// TwinCAT 3 PLC project PLC
// ProgramVersion: 3.1.4024.0
// libraries:
//   Tc2_Standard, * (Beckhoff Automation GmbH)
//   Tc2_System, * (Beckhoff Automation GmbH)
//   Tc3_Module, * (Beckhoff Automation GmbH)
// project tree:
//   / PlcTask.TcTTO
//   POUs/ MAIN.TcPOU, TankControl01.TcPOU, TankControl02.TcPOU
//   POUs/Simulation/ IntegralCalculate.TcPOU, Scale.TcPOU, Simulation.TcPOU, TankLevelSimulator.TcPOU
// real-time tasks:
//   TASK PlcTask: cycle T#10ms, priority 20, ADS port 350

CONFIGURATION PLC
    RESOURCE PLC ON TwinCAT3
        TASK PlcTask(INTERVAL := T#10ms, PRIORITY := 20);
        PROGRAM MAIN WITH PlcTask : MAIN;
    END_RESOURCE
END_CONFIGURATION

// ---- POUs/MAIN.TcPOU
PROGRAM MAIN
VAR
	TankControl01				: TankControl01;
	Enable						: BOOL;
	TempReq						: REAL := 22.0;
	VolReq						: REAL := 1.2;
	TankDiam					: REAL := 1.0;
	TankHeight					: REAL := 10;
	LevelSensor					: WORD;
	TempSensor					: WORD;
	StartControl				: BOOL;
	FillValve					: BOOL;
	EmptyValve					: BOOL;
	HeatValve					: BOOL;
	
	Temp						: REAL;
	MixerMotor: BOOL;
END_VAR

Simulation(TankDiam := TankDiam, FillValve := TankControl01.FillValveCmd, HeatValve := TankControl01.HeatValveCmd, EmptyValve := TankControl01.EmptyValveCmd);
TankControl01(
    Enable := Enable,
    TemperatureReq := TempReq,
    VolumeReq := VolReq,
    TankDiameter := TankDiam,
    TankHeight := TankHeight,
    LevelSensor := TO_WORD(Simulation.Level),
    TemperatureSensor := TO_WORD(Simulation.Temperature),
    StartControl := StartControl);
FillValve := TankControl01.FillValveCmd;
EmptyValve := TankControl01.EmptyValveCmd;
HeatValve := TankControl01.HeatValveCmd;
MixerMotor := TankControl01.MixerMotorCmd;
// LevelSensor: input not connected
// TempSensor: input not connected

END_PROGRAM

// ---- POUs/TankControl01.TcPOU
FUNCTION_BLOCK TankControl01
VAR_INPUT
	Enable				:	BOOL;		// enable
	TemperatureReq		:	REAL;		// temperature request
	VolumeReq			:	REAL;		// volume request
	TankDiameter		:	REAL;		
	TankHeight			:	REAL;
	LevelSensor			:	WORD;		// raw value from AI
	TemperatureSensor	:	WORD;		// raw value from AI
	StartControl		:	BOOL;		// start tank control
END_VAR
VAR_OUTPUT
	FillValveCmd		:	BOOL;		// valve to fill the tank
	EmptyValveCmd		:	BOOL;		// valve to empty the tank
	HeatValveCmd		:	BOOL;		// valve to heat the tank
	MixerMotorCmd		:	BOOL;		// mixer motor inside tank
END_VAR
VAR
	LevelScaled			: 	REAL;
	TemperatureScaled	: 	REAL;
	TankVolume			: 	REAL;
	CalculationsOK		:	BOOL;
	SeqStep				:	(START, FILL, HEAT, EMPTY) := START;
END_VAR

(*
When Start Control switch is activated , Fill Valve opens and liquid fills the tank.
When liquid reaches the requested level, Fill Valve closes. 
Then Heat Valve opens and heats up the liquid. 
When the liquid inside the tank reaches the requested temperature, Empty Valve opens to empty the tank.
Mixer Motor ensures stirring during the heating process.
*)

IF Enable THEN
	SetSequence();
	SetOutput();
END_IF

METHOD Calculations : BOOL
VAR_INPUT

END_VAR

VAR
	HeightTotal			: REAL;
	LevelDoneOk			: BOOL;
	VolumeDoneOk		: BOOL;
	TemperatureDoneOk	: BOOL;
END_VAR

VAR_OUTPUT
	DoneOk			: BOOL;			// conversion done OK
END_VAR
HeightTotal := TankDiameter + TankHeight;

LevelScaled := THIS^.Scale(Enable := TRUE,
			ValueIn := LevelSensor,
			ScaleInMin := 0,
			ScaleInMax := 65535,
			ScaleOutMin := 0,
			ScaleOutMax := HeightTotal,
			DoneOk =>LevelDoneOk);
			
TankVolume := THIS^.TankVolumeCalculate(Diameter := TankDiameter,
						  Height := TankHeight,
						  Level := LevelScaled,
						  DoneOk =>VolumeDoneOk);
						  
TemperatureScaled := THIS^.Scale(Enable := TRUE,
			ValueIn := TemperatureSensor,
			ScaleInMin := 0,
			ScaleInMax := 65535,
			ScaleOutMin := 0,
			ScaleOutMax := 100,
			DoneOk =>TemperatureDoneOk);
			
DoneOk := LevelDoneOk AND VolumeDoneOk AND TemperatureDoneOk;
END_METHOD

METHOD Scale : REAL
VAR_INPUT
	Enable			:	BOOL;		// enable function
	ValueIn			:	REAL;		// value to be scaled
	ScaleInMin		:	REAL;		// ScaleInMin, must be < then ScaleInMax
	ScaleInMax		:	REAL;		// ScaleInMax, must be > then ScaleInMin
	ScaleOutMin		:	REAL;		// ScaleOutMin, must be < then ScaleOutMax
	ScaleOutMax		:	REAL;		// ScaleOutMax, must be > then ScaleOutMin
END_VAR

VAR
	Error			:	BOOL;		// wrong input parameter
	Slope			:	REAL;
	Offset			:	REAL;
END_VAR

VAR_OUTPUT
	DoneOk			: BOOL;			// conversion done OK
END_VAR
IF Enable THEN
	IF 	ScaleOutMin >= ScaleOutMax OR 
		ScaleInMin >= ScaleInMax OR
		ValueIn < ScaleInMin OR 
		ValueIn > ScaleInMax THEN
		Error := TRUE;
	END_IF
	
	IF NOT Error THEN
		Slope 	:= (ScaleOutMax - ScaleOutMin) / (ScaleInMax - ScaleInMin);
		Offset 	:= ScaleOutMax - (Slope * ScaleInMax);
		DoneOk 	:= TRUE;
		Scale := (Slope * ValueIn) + Offset;
	ELSE
		DoneOk 	:= FALSE;
	END_IF
	
END_IF
END_METHOD

METHOD SetOutput : BOOL
VAR_INPUT
END_VAR
VAR_INST // added by the converter: edge detectors and wires of the graphical bodies
    _w1 : BOOL;
END_VAR
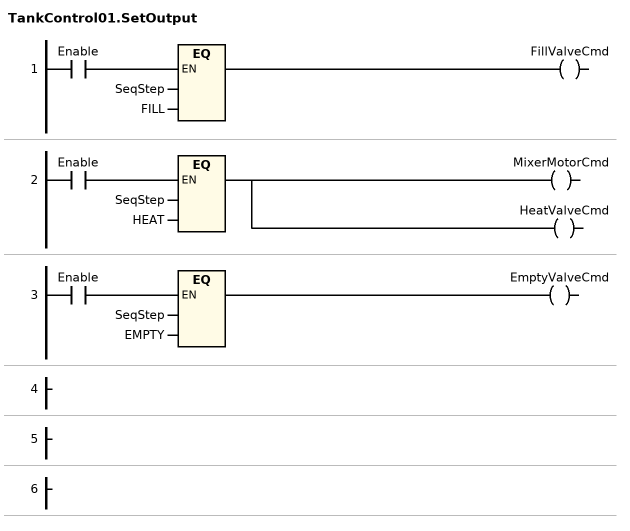
// NETWORK 1
FillValveCmd := Enable AND SeqStep = FILL;

// NETWORK 2
_w1 := Enable AND SeqStep = HEAT;
MixerMotorCmd := _w1;
HeatValveCmd := _w1;

// NETWORK 3
EmptyValveCmd := Enable AND SeqStep = EMPTY;

// NETWORK 4

// NETWORK 5

// NETWORK 6
END_METHOD

METHOD SetSequence : BOOL
VAR_INPUT
END_VAR
Calculations(DoneOk=>CalculationsOK);

IF CalculationsOK AND SeqStep = START AND StartControl THEN
	SeqStep := FILL;
ELSIF CalculationsOK AND SeqStep = FILL AND TankVolume>VolumeReq THEN
	SeqStep := HEAT;
ELSIF CalculationsOK AND SeqStep = HEAT AND TemperatureScaled > TemperatureReq THEN
	SeqStep := EMPTY;
ELSIF CalculationsOK AND SeqStep = EMPTY AND TankVolume < 0.001 THEN
	SeqStep := START;
END_IF
END_METHOD

METHOD TankVolumeCalculate : REAL
VAR_INPUT
	Diameter			:	REAL;		// tank diameter
	Height				:	REAL;		// tank height
	Level				:	REAL;		// current level measured
END_VAR

VAR
	LevelRadius			:	REAL;		// level radius in circle
	Volume				:	REAL;		// volume
END_VAR

VAR_OUTPUT
	DoneOk			: BOOL;				// conversion done OK
END_VAR
// check level depth
IF Level < 0 THEN
	Level := 0;	
END_IF

// check level height - tank cannot be overfilled
IF Level > (Diameter/2 + Height) THEN
	Level := Diameter/2 + Height;
END_IF


// hemisphere
IF Level <= Diameter/2 THEN
	// hemisphere partially filled
	LevelRadius := SQRT(Level * (Diameter/2 - Level));
	Volume := (TO_REAL(PI)/6) * Level * (3 * LevelRadius * LevelRadius + Level * Level);
ELSE
	// hemisphere filled
	Volume := 2.0/3.0 * TO_REAL(PI) * Diameter/2 * Diameter/2 * Diameter/2;
END_IF

// something in the cylinder
IF Level > Diameter/2 THEN
	Volume := Volume + (Level - Diameter/2) * TO_REAL(PI) * Diameter/2 * Diameter/2;
END_IF

TankVolumeCalculate := Volume;
DoneOk := TRUE;
END_METHOD

END_FUNCTION_BLOCK

// ---- POUs/Simulation/Scale.TcPOU
FUNCTION Scale : REAL
VAR_INPUT
	Enable			:	BOOL;		// enable function
	ValueIn			:	REAL;		// value to be scaled
	ScaleInMin		:	REAL;		// ScaleInMin, must be < then ScaleInMax
	ScaleInMax		:	REAL;		// ScaleInMax, must be > then ScaleInMin
	ScaleOutMin		:	REAL;		// ScaleOutMin, must be < then ScaleOutMax
	ScaleOutMax		:	REAL;		// ScaleOutMax, must be > then ScaleOutMin
END_VAR
VAR
	Error			:	BOOL;		// wrong input parameter
	Slope			:	REAL;
	Offset			:	REAL;
END_VAR

VAR_OUTPUT
	DoneOk			: BOOL;			// conversion done OK
END_VAR

IF Enable THEN
	IF 	ScaleOutMin >= ScaleOutMax OR 
		ScaleInMin >= ScaleInMax OR
		ValueIn < ScaleInMin OR 
		ValueIn > ScaleInMax THEN
		Error := TRUE;
	END_IF
	
	IF NOT Error THEN
		Slope 	:= (ScaleOutMax - ScaleOutMin) / (ScaleInMax - ScaleInMin);
		Offset 	:= ScaleOutMax - (Slope * ScaleInMax);
		DoneOk 	:= TRUE;
		Scale := (Slope * ValueIn) + Offset;
	ELSE
		DoneOk 	:= FALSE;
	END_IF
	
END_IF

END_FUNCTION

// ---- POUs/Simulation/Simulation.TcPOU
PROGRAM Simulation
VAR_INPUT
	TankDiam					:	REAL;
	FillValve					:	BOOL;
	HeatValve					:	BOOL;
	EmptyValve					:	BOOL;
END_VAR


VAR
		TankLevelSimulator		: 	TankLevelSimulator;
		Flow					:	REAL;
		TemperatureSim			: 	REAL;
		
END_VAR

VAR_OUTPUT
		Level					:	REAL;
		Temperature				:	REAL;
END_VAR

// flow depending on valve position
Flow := TO_REAL(FillValve) * 0.1 - TO_REAL(EmptyValve) * 0.05;

TankLevelSimulator(	Flow:=Flow,
					TankDiameter:=TankDiam
					);
					

Level := Scale(
				Enable:=TRUE , 
				ValueIn:=TankLevelSimulator.Level , 
				ScaleInMin:= 0, 
				ScaleInMax:= 50, 
				ScaleOutMin:= 0, 
				ScaleOutMax:= 65535, 
				DoneOk=> );
				
// temperature depending on valve position
IF HeatValve THEN
	TemperatureSim := TemperatureSim + 0.002;
ELSIF NOT HeatValve AND Temperature > 0 THEN
	TemperatureSim := TemperatureSim - 0.002;
END_IF

Temperature := Scale(
					Enable:=TRUE , 
					ValueIn:=TemperatureSim , 
					ScaleInMin:= 0, 
					ScaleInMax:= 40, 
					ScaleOutMin:= 0, 
					ScaleOutMax:= 65535, 
					DoneOk=> );

END_PROGRAM

// ---- POUs/Simulation/TankLevelSimulator.TcPOU
FUNCTION_BLOCK TankLevelSimulator
VAR_INPUT
	Flow				:	REAL;				// input flow in [m3/s]
	TankDiameter		:	REAL;				// tank diameter in [m]
END_VAR
VAR_OUTPUT
	Level				:	REAL;				// output tank level in [m]
END_VAR
VAR
	TankArea			:	REAL;				// tank cross section area in [m2]
	Integral			:	IntegralCalculate;	// integral calculation
END_VAR

// tank cross area
TankArea := TO_REAL(PI) *(TankDiameter * TankDiameter / 4.0 );


IF Level>=0 AND TankArea<>0 THEN
	Integral(InputValue:=(Flow - (0.001 * SQRT(Level))) / TankArea);
	Level := Integral.IntegratedValue;
	IF Level < 0 THEN
		Level := 0;
	END_IF
END_IF

END_FUNCTION_BLOCK

// ---- POUs/Simulation/IntegralCalculate.TcPOU
FUNCTION_BLOCK IntegralCalculate
VAR_INPUT
	InputValue 		: REAL;
	PlcCycleTime 	: REAL := 0.01;
END_VAR
VAR_OUTPUT
	    IntegratedValue : REAL := 0.0;
END_VAR
VAR
	PrevInputValue : REAL := 0.0;
END_VAR

// Integration logic (Trapezoidal Method)
IntegratedValue := IntegratedValue + ((InputValue + PrevInputValue) * 0.5 * PlcCycleTime);

// Update previous value for next cycle
PrevInputValue := InputValue;

END_FUNCTION_BLOCK

// ---- POUs/TankControl02.TcPOU
FUNCTION_BLOCK TankControl02
VAR_INPUT
	Enable				:	BOOL;		// enable
	TemperatureReq		:	REAL;		// temperature request
	VolumeReq			:	REAL;		// volume request
	TankDiameter		:	REAL;		
	TankHeight			:	REAL;
	LevelSensor			:	WORD;		// raw value from AI
	TemperatureSensor	:	WORD;		// raw value from AI
	StartControl		:	BOOL;		// start tank control
END_VAR
VAR_OUTPUT
	FillValveCmd		:	BOOL;		// valve to fill the tank
	EmptyValveCmd		:	BOOL;		// valve to empty the tank
	HeatValveCmd		:	BOOL;		// valve to heat the tank
	MixerMotorCmd		:	BOOL;		// mixer motor inside tank
END_VAR
VAR
	LevelScaled			: 	REAL;
	TemperatureScaled	: 	REAL;
	TankVolume			: 	REAL;
	CalculationsOK		:	BOOL;
	SeqStep				:	(START, FILL, HEAT, EMPTY) := START;
END_VAR

(*
When Start Control switch is activated , Fill Valve opens and liquid fills the tank.
When liquid reaches the requested level, Fill Valve closes. 
Then Heat Valve opens and heats up the liquid. 
When the liquid inside the tank reaches the requested temperature, Empty Valve opens to empty the tank.
Mixer Motor ensures stirring during the heating process.
*)

IF Enable THEN
	SetSequence();
	SetOutput();
END_IF

METHOD Calculations : BOOL
VAR_INPUT

END_VAR

VAR
	HeightTotal			: REAL;
	LevelDoneOk			: BOOL;
	VolumeDoneOk		: BOOL;
	TemperatureDoneOk	: BOOL;
END_VAR

VAR_OUTPUT
	DoneOk			: BOOL;			// conversion done OK
END_VAR
HeightTotal := TankDiameter + TankHeight;

LevelScaled := THIS^.Scale(Enable := TRUE,
			ValueIn := LevelSensor,
			ScaleInMin := 0,
			ScaleInMax := 65535,
			ScaleOutMin := 0,
			ScaleOutMax := HeightTotal,
			DoneOk =>LevelDoneOk);
			
TankVolume := THIS^.TankVolumeCalculate(Diameter := TankDiameter,
						  Height := TankHeight,
						  Level := LevelScaled,
						  DoneOk =>VolumeDoneOk);
						  
TemperatureScaled := THIS^.Scale(Enable := TRUE,
			ValueIn := TemperatureSensor,
			ScaleInMin := 0,
			ScaleInMax := 65535,
			ScaleOutMin := 0,
			ScaleOutMax := 100,
			DoneOk =>TemperatureDoneOk);
			
DoneOk := LevelDoneOk AND VolumeDoneOk AND TemperatureDoneOk;
END_METHOD

METHOD Scale : REAL
VAR_INPUT
	Enable			:	BOOL;		// enable function
	ValueIn			:	REAL;		// value to be scaled
	ScaleInMin		:	REAL;		// ScaleInMin, must be < then ScaleInMax
	ScaleInMax		:	REAL;		// ScaleInMax, must be > then ScaleInMin
	ScaleOutMin		:	REAL;		// ScaleOutMin, must be < then ScaleOutMax
	ScaleOutMax		:	REAL;		// ScaleOutMax, must be > then ScaleOutMin
END_VAR

VAR
	Error			:	BOOL;		// wrong input parameter
	Slope			:	REAL;
	Offset			:	REAL;
END_VAR

VAR_OUTPUT
	DoneOk			: BOOL;			// conversion done OK
END_VAR
IF Enable THEN
	IF 	ScaleOutMin >= ScaleOutMax OR 
		ScaleInMin >= ScaleInMax OR
		ValueIn < ScaleInMin OR 
		ValueIn > ScaleInMax THEN
		Error := TRUE;
	END_IF
	
	IF NOT Error THEN
		Slope 	:= (ScaleOutMax - ScaleOutMin) / (ScaleInMax - ScaleInMin);
		Offset 	:= ScaleOutMax - (Slope * ScaleInMax);
		DoneOk 	:= TRUE;
		Scale := (Slope * ValueIn) + Offset;
	ELSE
		DoneOk 	:= FALSE;
	END_IF
	
END_IF
END_METHOD

METHOD SetOutput : BOOL
VAR_INPUT
END_VAR
IF Enable THEN
	MixerMotorCmd:=FALSE;
	FillValveCmd:=FALSE;
	HeatValveCmd:=FALSE;
	EmptyValveCmd:=FALSE;
	
	CASE SeqStep OF
		FILL:		FillValveCmd:=TRUE;	

		HEAT:		MixerMotorCmd:=TRUE;
					HeatValveCmd:=TRUE;
		
		EMPTY:		EmptyValveCmd:=TRUE;	
	END_CASE
END_IF
END_METHOD

METHOD SetSequence : BOOL
VAR_INPUT
END_VAR
Calculations(DoneOk=>CalculationsOK);

IF CalculationsOK AND SeqStep = START AND StartControl THEN
	SeqStep := FILL;
ELSIF CalculationsOK AND SeqStep = FILL AND TankVolume>VolumeReq THEN
	SeqStep := HEAT;
ELSIF CalculationsOK AND SeqStep = HEAT AND TemperatureScaled > TemperatureReq THEN
	SeqStep := EMPTY;
ELSIF CalculationsOK AND SeqStep = EMPTY AND TankVolume < 0.001 THEN
	SeqStep := START;
END_IF
END_METHOD

METHOD TankVolumeCalculate : REAL
VAR_INPUT
	Diameter			:	REAL;		// tank diameter
	Height				:	REAL;		// tank height
	Level				:	REAL;		// current level measured
END_VAR

VAR
	LevelRadius			:	REAL;		// level radius in circle
	Volume				:	REAL;		// volume
END_VAR

VAR_OUTPUT
	DoneOk			: BOOL;				// conversion done OK
END_VAR
// check level depth
IF Level < 0 THEN
	Level := 0;	
END_IF

// check level height - tank cannot be overfilled
IF Level > (Diameter/2 + Height) THEN
	Level := Diameter/2 + Height;
END_IF


// hemisphere
IF Level <= Diameter/2 THEN
	// hemisphere partially filled
	LevelRadius := SQRT(Level * (Diameter/2 - Level));
	Volume := (TO_REAL(PI)/6) * Level * (3 * LevelRadius * LevelRadius + Level * Level);
ELSE
	// hemisphere filled
	Volume := 2.0/3.0 * TO_REAL(PI) * Diameter/2 * Diameter/2 * Diameter/2;
END_IF

// something in the cylinder
IF Level > Diameter/2 THEN
	Volume := Volume + (Level - Diameter/2) * TO_REAL(PI) * Diameter/2 * Diameter/2;
END_IF

TankVolumeCalculate := Volume;
DoneOk := TRUE;
END_METHOD

END_FUNCTION_BLOCK
